INTERFACE I_Resettable EXTENDS I_Base

METHOD Reset
END_METHOD

END_INTERFACE

(* stored: Version 1.1.0.1, ProductVersion 3.1.4026.18
   Itf I_Resettable: Id {b6038dde-a86b-4107-a048-b4750546394b}
   Method Reset: Id {03c44dbf-19ea-45ce-8aee-0335a91d1808} *)
